FUNCTION_BLOCK HPU
VAR_INPUT
	par : ST_pValveControlledCylinder;
END_VAR
VAR_OUTPUT
	TankPressure : LREAL;
	SupplyPressure : LREAL;
END_VAR
VAR
	//Pump
	fbPump : Pump;
	PumpTorque : LREAL;
	PumpFlowRate : LREAL;
END_VAR


//Pump
fbPump(
MotorSpeedRPM := 413.2,
PumpDisplacement := 10.6E-6,
DeltaMaxPressure := 250.0,
PumpTorque => PumpTorque,
PumpFlowRate => PumpFlowRate
);

TankPressure := 1.2E5;
SupplyPressure := 180E5; 

G_ActuationSystems.ReturnPressure := TankPressure;
G_ActuationSystems.SupplyPressure := SupplyPressure;

END_FUNCTION_BLOCK

(* stored: Version 1.1.0.1, ProductVersion 3.1.4024.9
   POU HPU: Id {91e109f3-38cc-4845-95f1-12a5ba54273f}, SpecialFunc None *)
